FUNCTION_BLOCK PUBLIC PAFExtruding EXTENDS PARoutingFunction
VAR_INPUT
END_VAR
VAR_OUTPUT
END_VAR
VAR
	_ACMethod : ACMethodExtruding;
END_VAR

PROPERTY ACMethod : IACMethod
GET
ACMethod := _ACMethod;
END_GET
END_PROPERTY

END_FUNCTION_BLOCK

(* stored: Version 1.1.0.1, ProductVersion 3.1.4020.12
   POU PAFExtruding: Id {f1e5dd8c-da1b-4836-97e3-8dc2981d9e48}, SpecialFunc None
   Property ACMethod: Id {4f1580cc-6142-4bf2-a910-eb019515bde2}
   Get Get: Id {8b9c93c1-0723-4de7-8b38-92f9487a07fc} *)
